(* PLC project SafeLOGIC-1, BrAutomation SafeDESIGNER  4.3.3.7 *)
(* stored: companyURL http://www.br-automation.com, creationDateTime Tue Jun 23 09:46:06 2020 *)

PROGRAM Output

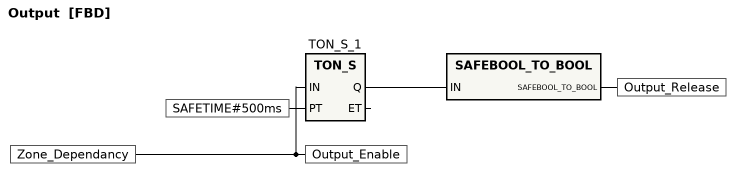
(* FBD diagram, written out as Structured Text *)
Output_Enable := Zone_Dependancy;
TON_S_1(IN := Zone_Dependancy, PT := SAFETIME#500ms);
Output_Release := SAFEBOOL_TO_BOOL(TON_S_1.Q);
END_PROGRAM
